FUNCTION_BLOCK FBCOMPARE
VAR_INPUT
END_VAR
VAR_OUTPUT
END_VAR
VAR
END_VAR

END_FUNCTION_BLOCK

(* stored: Version 1.1.0.1, ProductVersion 3.1.4026.18
   POU FBCOMPARE: Id {87c16756-fddf-42f9-a69c-1419ae458759}, SpecialFunc None *)
